SYSTEM X2Y2_TESTL (* Local Multicast Configuration to test X2Y2 *)
  (* Standard: 61499-1 *)
  (* Version 0.0, 2003-08-11, JHC, Rockwell Automation, Adapted from TESTD_X2Y2. *)
  APPLICATION APP1 (* Testing FB_X2Y2 *)
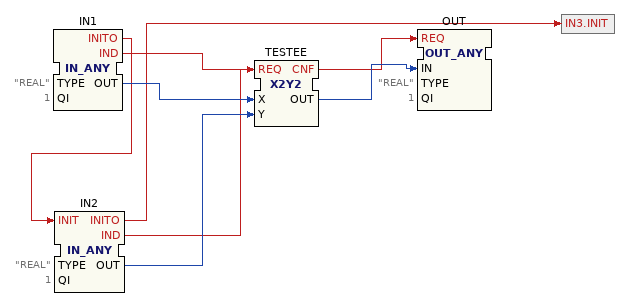
    FBS
      IN1 : IN_ANY(TYPE := "REAL", QI := 1);
      IN2 : IN_ANY(TYPE := "REAL", QI := 1);
      TESTEE : X2Y2;
      OUT : OUT_ANY(TYPE := "REAL", QI := 1);
    END_FBS
    EVENT_CONNECTIONS
      IN1.INITO TO IN2.INIT;
      IN2.INITO TO IN3.INIT;
      IN1.IND TO TESTEE.REQ;
      IN2.IND TO TESTEE.REQ;
      TESTEE.CNF TO OUT.REQ;
    END_CONNECTIONS
    DATA_CONNECTIONS
      IN1.OUT TO TESTEE.X;
      IN2.OUT TO TESTEE.Y;
      TESTEE.OUT TO OUT.IN;
    END_CONNECTIONS
  END_APPLICATION
  DEVICE DEV1 : FRAME_DEVICE(BOUNDS := [150,150,125,100], GRID := [1,1])
    RESOURCE RES1 : PANEL_RESOURCE
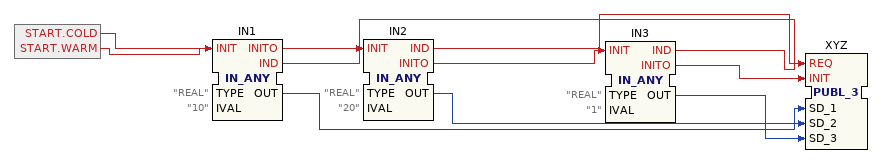
      FBS
        IN1 : IN_ANY(TYPE := "REAL", IVAL := "10");
        IN2 : IN_ANY(TYPE := "REAL", IVAL := "20");
        XYZ : PUBL_3;
        IN3 : IN_ANY(TYPE := "REAL", IVAL := "1");
      END_FBS
      EVENT_CONNECTIONS
        START.COLD TO IN1.INIT;
        START.WARM TO IN1.INIT;
        IN1.INITO TO IN2.INIT;
        IN1.IND TO XYZ.REQ;
        IN2.IND TO XYZ.REQ;
        IN2.INITO TO IN3.INIT;
        IN3.IND TO XYZ.REQ;
        IN3.INITO TO XYZ.INIT;
      END_CONNECTIONS
      DATA_CONNECTIONS
        IN1.OUT TO XYZ.SD_1;
        IN2.OUT TO XYZ.SD_2;
        IN3.OUT TO XYZ.SD_3;
      END_CONNECTIONS
    END_RESOURCE
  END_DEVICE
  DEVICE DEV2 : FRAME_DEVICE(BOUNDS := [150,250,125,75], GRID := [1,1])
    RESOURCE RES2 : PANEL_RESOURCE
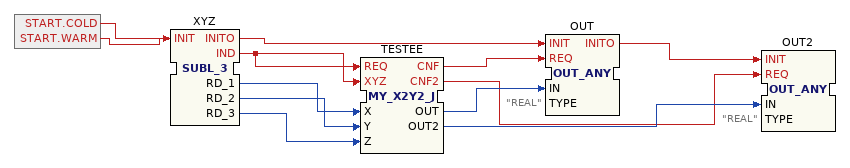
      FBS
        XYZ : SUBL_3;
        TESTEE : MY_X2Y2_J;
        OUT : OUT_ANY(TYPE := "REAL");
        OUT2 : OUT_ANY(TYPE := "REAL");
      END_FBS
      EVENT_CONNECTIONS
        START.COLD TO XYZ.INIT;
        START.WARM TO XYZ.INIT;
        XYZ.INITO TO OUT.INIT;
        XYZ.IND TO TESTEE.REQ;
        TESTEE.CNF TO OUT.REQ;
        OUT.INITO TO OUT2.INIT;
        TESTEE.CNF2 TO OUT2.REQ;
        XYZ.IND TO TESTEE.XYZ;
      END_CONNECTIONS
      DATA_CONNECTIONS
        TESTEE.OUT TO OUT.IN;
        XYZ.RD_1 TO TESTEE.X;
        XYZ.RD_2 TO TESTEE.Y;
        XYZ.RD_3 TO TESTEE.Z;
        TESTEE.OUT2 TO OUT2.IN;
      END_CONNECTIONS
    END_RESOURCE
  END_DEVICE
  MAPPINGS
    APP1.IN1 ON DEV1.RES1.IN1;
    APP1.IN2 ON DEV1.RES1.IN2;
    APP1.TESTEE ON DEV2.RES2.TESTEE;
    APP1.OUT ON DEV2.RES2.OUT;
  END_MAPPINGS
END_SYSTEM
